TYPE ST_LaudaWriteCommands_Cooling :
STRUCT
	CoolingMode	: STRING := 'OUT_SP_02';
END_STRUCT
END_TYPE

(* stored: Version 1.1.0.1, ProductVersion 3.1.4024.13
   DUT ST_LaudaWriteCommands_Cooling: Id {f8a0d94f-2c54-4965-bf92-c48614f8039f} *)
